DATA_BLOCK "CoolingTank_DB"
{ S7_Optimized_Access := 'TRUE' }
"FB_CoolingTank"


BEGIN

END_DATA_BLOCK
